// TIA Portal V17 export
// export: Created 2026-07-06T15:33:05.0629462Z, ExportSetting WithDefaults, DisplayName Totally Integrated Automation Portal, DisplayVersion V17, DisplayName TIA Portal Openness, DisplayVersion V17, DisplayName TIA Portal Version Control Interface, DisplayVersion V17, DisplayName STEP 7 Professional, DisplayVersion V17, DisplayName STEP 7 Safety, DisplayVersion V17, DisplayName WinCC Professional, DisplayVersion V17
VAR_GLOBAL   // PLC tag table "Default tag table"
   System_Byte AT %MB1 : Byte;
   FirstScan AT %M1.0 : Bool;
   DiagStatusUpdate AT %M1.1 : Bool;
   AlwaysTRUE AT %M1.2 : Bool;
   AlwaysFALSE AT %M1.3 : Bool;
   Clock_Byte AT %MB0 : Byte;
   Clock_10Hz AT %M0.0 : Bool;
   Clock_5Hz AT %M0.1 : Bool;
   "Clock_2.5Hz" AT %M0.2 : Bool;
   Clock_2Hz AT %M0.3 : Bool;
   "Clock_1.25Hz" AT %M0.4 : Bool;
   Clock_1Hz AT %M0.5 : Bool;
   "Clock_0.625Hz" AT %M0.6 : Bool;
   "Clock_0.5Hz" AT %M0.7 : Bool;
   BMS_Connect_req AT %M2.0 : Bool;
   Send_data AT %M2.2 : Bool;
   Kinco_connect_req AT %M2.1 : Bool;
   Node_ID_1 AT %MW4 : Int;
   Node_ID_2 AT %MW6 : Int;
   Connection_Established AT %M2.3 : Bool;
   Motor_1_Select_mode AT %MB3 : Byte;
   move_data_pulse AT %M2.4 : Bool;
   motor_1_control_word AT %MW10 : Word;
   LH_pulse_out AT %M2.6 : Bool;
   RH_pulse_out AT %M2.7 : Bool;
   RH_Speed AT %MD18 : DInt;
   LH_Speed AT %MD22 : DInt;
   send_data_pulse AT %M2.5 : Bool;
   node_terminate AT %I0.0 : Bool;
   motor_1_target_rpm AT %MD12 : DInt;
   motor_1_target_pos AT %MD28 : DInt;
   motor_1_profile_speed AT %MD32 : DInt;
   Tag_1 AT %I0.2 : Bool;
   wake_node_trigger AT %I0.1 : Bool;
   Motor_2_Select_mode AT %MB8 : Byte;
   motor_2_control_word AT %MW16 : Word;
   motor_2_target_rpm AT %MD36 : DInt;
   motor_2_target_pos AT %MD40 : DInt;
   motor_2_profile_speed AT %MD44 : DInt;
END_VAR
